// TIA Portal V18 export
// export: Created 2026-06-08T16:32:20.9312348Z, ExportSetting WithDefaults, DisplayName Totally Integrated Automation Portal, DisplayVersion V18, DisplayName TIA Portal Openness, DisplayVersion V18, DisplayName TIA Portal Version Control Interface, DisplayVersion V18, DisplayName STEP 7 Professional, DisplayVersion V18, DisplayName STEP 7 Safety, DisplayVersion V18, DisplayName WinCC Professional, DisplayVersion V18
DATA_BLOCK "base_production_fb_DB"   // DB17
VERSION : 0.1
// stored: AutoNumber true, InstanceOfName base_production_fb, InstanceOfType FB
"base_production_fb"
BEGIN
END_DATA_BLOCK
